TYPE MoverComSubscribe :
STRUCT
  Request : MoverComRequest; // contains booleans that are used to start a specific sequence.
  Equipment : MoverComSubscribeEquipment;  // structs for equipment objects which are used by the bridges
END_STRUCT
END_TYPE

(* stored: Version 1.1.0.1
   DUT MoverComSubscribe: Id {5f1c210f-6015-4761-9977-57c9f281606e} *)
